// TwinCAT 3 PLC project CollectionTests
// ProgramVersion: 3.1.4026.19
// libraries:
//   AbstractObjectTestLib, * (ekvip automation GmbH)
//   CNM_AbstractObject, * (ekvip automation GmbH)
//   CNM_CollectionInterfaces, * (ekvip automation GmbH)
//   CNM_Collections, * (ekvip automation GmbH)
//   CNM_CollectionTestLib, * (ekvip automation GmbH)
//   CNM_ReturnTypes, * (ekvip automation GmbH)
//   Tc2_Standard, * (Beckhoff Automation GmbH)
//   Tc2_System, * (Beckhoff Automation GmbH)
//   Tc3_Module, * (Beckhoff Automation GmbH)
//   TcUnit, * (www.tcunit.org)
// project tree:
//   / PlcTask.TcTTO
//   POUs/ArrayListSorter/ ContainerBasedArrayListSorterTest.TcPOU, TestArrayList.TcPOU
//   POUs/BBSTrees/ concretBBSTreeTest.TcPOU, TreeTestClass.TcPOU
//   POUs/LinkedList/ LinkedListTest.TcPOU, TestLinkedList.TcPOU
//   POUs/ MAIN.TcPOU
// real-time tasks:
//   TASK PlcTask: cycle T#100us, priority 20, ADS port 350

CONFIGURATION CollectionTests
    RESOURCE PLC ON TwinCAT3
        TASK PlcTask(INTERVAL := T#100us, PRIORITY := 20);
        PROGRAM MAIN WITH PlcTask : MAIN;
    END_RESOURCE
END_CONFIGURATION

// ---- POUs/MAIN.TcPOU
PROGRAM MAIN
VAR
	optionVerbose 						:BOOL := FALSE;
    testCollectionFactory 				:CNM_Collections.CollectionFactory();
	
	
	(*Linked List Tests*)
	linkedList 							:CNM_Collections.LinkedList();
	linkedList2 						:CNM_Collections.LinkedList();
	linkedList3							:CNM_Collections.LinkedList();
	LinkedListTest 						:CNM_CollectionTestLib.ListInterfaceTest(linkedList, linkedList2, testCollectionFactory);
	linkedListDispatcher				:CNM_CollectionTestLib.ListDispatcher(linkedList3);
	linkedListCollectionTest			:CNM_CollectionTestLib.CollectionInterfaceTest(linkedList3, testCollectionFactory, linkedListDispatcher);
	LinkedListObjectTest  				:AbstractObject_Test(linkedList, linkedList2);
	LinkedListTest2						:LinkedListTest(linkedList, linkedList2, testCollectionFactory);
	linkedListForIteratorTest			:CNM_Collections.LinkedList();
	forwardLinkedListIterator			:CNM_Collections.ForwardLinkedListIterator(list:=linkedListForIteratorTest);
	inverseLinkedListIterator			:CNM_Collections.InverseLinkedListIterator(list:=linkedListForIteratorTest);
	linkedListDispatcherIteratorTest	:CNM_CollectionTestLib.ListDispatcher(linkedListForIteratorTest);
	linkedListForwardIteratorTest		:CNM_CollectionTestLib.IteratorInterfaceTest(linkedListForIteratorTest,forwardLinkedListIterator,linkedListDispatcherIteratorTest);
	linkedListInverseIteratorTest		:CNM_CollectionTestLib.IteratorInterfaceTest(linkedListForIteratorTest,inverseLinkedListIterator,linkedListDispatcherIteratorTest);
	
	(*Linkedlistsorter Tests*)
	(*Mergesorter*)
	LinkedListMergeSorter1				:CNM_Collections.LinkedListMergeSorter();
	LinkedListMergeSorter2				:CNM_Collections.LinkedListMergeSorter();
	LinkedListMergeSorterTest			:CNM_CollectionTestLib.ListSorterTest(ListFactory := testCollectionFactory, externListSorter := LinkedListMergeSorter1, verboseLogging := optionVerbose);
	LinkedListMergeSorterObjectTest 	:AbstractObject_Test(LinkedListMergeSorter1, LinkedListMergeSorter2);
	
	(*Array List Tests*)
	arrayList1 							:CNM_Collections.ArrayList();
	arrayList2 							:CNM_Collections.ArrayList();
	arrayList3 							:CNM_Collections.ArrayList();	
	arrayList4							:CNM_Collections.ArrayList();
	ArrayListTest 						:CNM_CollectionTestLib.ListInterfaceTest(arrayList1, arrayList2, testCollectionFactory);
	arrayListDispatcher					:CNM_CollectionTestLib.ListDispatcher(arrayList3);		
	arrayListCollectionTest				:CNM_CollectionTestLib.CollectionInterfaceTest(arrayList3, testCollectionFactory, arrayListDispatcher);
	arrayListIndexableTest 				:CNM_CollectionTestLib.IndexableCollectionTest(arrayList4);
	arrayListObjectTest  				:AbstractObject_Test(arrayList1, arrayList2);
	arrayListForIteratorTest			:CNM_Collections.ArrayList();
	forwardArrayListIterator			:CNM_Collections.ForwardArrayListIterator(arrayList:=arrayListForIteratorTest);
	inverseArrayListIterator			:CNM_Collections.InverseArrayListIterator(arrayList:=arrayListForIteratorTest);
	arrayListDispatcherIteratorTest		:CNM_CollectionTestLib.ListDispatcher(arrayListForIteratorTest);
	arrayListForwardIteratorTest		:CNM_CollectionTestLib.IteratorInterfaceTest(arrayListForIteratorTest,forwardArrayListIterator,arrayListDispatcherIteratorTest);
	arrayListInverseIteratorTest		:CNM_CollectionTestLib.IteratorInterfaceTest(arrayListForIteratorTest,inverseArrayListIterator,arrayListDispatcherIteratorTest);
	
	(*Arraylistsorter Tests*)
	(*Mergesorter*)
	ArrayListMergeSorter1 				:CNM_Collections.ArrayListMergeSorter();
	ArrayListMergeSorter2 				:CNM_Collections.ArrayListMergeSorter();
	ArrayListMergeSorterTest 			:ContainerBasedArrayListSorterTest(ListFactory := testCollectionFactory, externListSorter := ArrayListMergeSorter1, verboseLogging := optionVerbose);
	ArrayListMergeSorterObjectTest 		:AbstractObject_Test(ArrayListMergeSorter1, ArrayListMergeSorter2);
	
	(*Timsorter*)
	ArrayListTwinSorter 				:CNM_Collections.ArrayListTwinSorter();
	ArrayListTwinSorter2 				:CNM_Collections.ArrayListTwinSorter(); 
	ArrayListTwinSorterTest 				:ContainerBasedArrayListSorterTest(ListFactory:=testCollectionFactory,externListSorter := ArrayListTwinSorter, verboseLogging := optionVerbose);
	ArrayListTwinSorterObjectTest 		:AbstractObjectTestLib.AbstractObject_Test(ArrayListTwinSorter, ArrayListTwinSorter2);
	
	(*Shellsorter*)
	ArrayListShellSorter 				:CNM_Collections.ArrayListShellSorter;
	ArrayListShellSorter2 				:CNM_Collections.ArrayListShellSorter;
	ArrayListShellSorterTest 			:ContainerBasedArrayListSorterTest(ListFactory:=testCollectionFactory,externListSorter := ArrayListShellSorter, verboseLogging := optionVerbose);
	ArrayListShellSorterObjectTest 		:AbstractObjectTestLib.AbstractObject_Test(ArrayListShellSorter, ArrayListShellSorter2);

	(*Treetests*)
	TreeFactory							:CNM_Collections.CollectionFactory();
	InterfaceTreeTest					:CNM_CollectionTestLib.BalancedBinaryTreeTest(Treefactory := Treefactory);
	ClassTreeTest						:concretBBSTreeTest(Treefactory := TreeFactory);
	tree1								:CNM_Collections.BalancedBinarySearchTree(0);
	tree2								:CNM_Collections.BalancedBinarySearchTree(0);
	tree3								:CNM_Collections.BalancedBinarySearchTree(0);
	treeDispatcher						:CNM_CollectionTestLib.TreeDispatcher(tree3);
	treeCollectionTest					:CNM_CollectionTestLib.CollectionInterfaceTest(tree3, treeFactory, treeDispatcher);
	objectTreeTest						:AbstractObject_Test(tree1, tree2);
	treeForIteratorTest					:CNM_Collections.BalancedBinarySearchTree(0);
	bfsTreeIterator						:CNM_Collections.BfsBbstIterator(tree:=treeForIteratorTest);
	dfsTreeIterator						:CNM_Collections.DfsBbstIterator(tree:=treeForIteratorTest);
	inorderTreeIterator					:CNM_Collections.InorderBbstIterator(tree:=treeForIteratorTest);
	treeDispatcherIteratorTest			:CNM_CollectionTestLib.TreeDispatcher(treeForIteratorTest);
	treeBFSIteratorTest					:CNM_CollectionTestLib.IteratorInterfaceTest(treeForIteratorTest,bfsTreeIterator,treeDispatcherIteratorTest);
	treeDFSIteratorTest					:CNM_CollectionTestLib.IteratorInterfaceTest(treeForIteratorTest,dfsTreeIterator,treeDispatcherIteratorTest);
	treeInorderIteratorTest				:CNM_CollectionTestLib.IteratorInterfaceTest(treeForIteratorTest,inorderTreeIterator,treeDispatcherIteratorTest);
END_VAR
VAR CONSTANT
	NOT_DEFINED 						:__XWORD := 0;
END_VAR

 TcUnit.RUN_IN_SEQUENCE();

END_PROGRAM

// ---- POUs/LinkedList/LinkedListTest.TcPOU
FUNCTION_BLOCK LinkedListTest EXTENDS CNM_CollectionTestLib.ListInterfaceTest;
VAR_INPUT
END_VAR
VAR_OUTPUT
END_VAR
VAR
END_VAR

THIS^.SortAndCheckPreviousElement('SortAndCheckElementPrevious');

METHOD FB_init : BOOL
VAR_INPUT
    bInitRetains : BOOL; // if TRUE, the retain variables are initialized (warm start / cold start)
    bInCopyCode : BOOL;  // if TRUE, the instance afterwards gets moved into the copy code (online change)
	(*main list to be tested*)
	emptyList1 :CNM_CollectionInterfaces.IList;
	(*secondary list to be tested for appendCollection test*)
	emptyList2 :CNM_CollectionInterfaces.IList;
	(*factory needed for forEach tests, not tested*)
	actionListFactory :CNM_CollectionInterfaces.ICollectionFactory;
END_VAR
THIS^.externalList := emptyList1;
THIS^.externalList2 := emptyList2;
THIS^.listFactory := actionListFactory;
END_METHOD

METHOD SortAndCheckPreviousElement
VAR_INPUT
	testInstanceIdentifier	:STRING(255);
END_VAR
VAR
	testname				:STRING(255);
	dequeuedElement			:CNM_AbstractObject.IObject;
	lastElement				:CNM_CollectionInterfaces.IDoublyLinkedElement;
	lastElementPrevious		:CNM_AbstractObject.IObject;
	foo						:CNM_AbstractObject.IObject;
	comparisonResult		:BOOL;
	index					:INT;
END_VAR
VAR_INST
	newLinkedList			:CNM_CollectionInterfaces.ILinkedList;
	specialList				:TestLinkedList;
	listToSort 				:CNM_CollectionInterfaces.IList;
	sortState				:CNM_ReturnTypes.SingleExecutionState;
	sortReady				:BOOL := FALSE;
	initSuccess				:BOOL := FALSE;
END_VAR
testname := Tc2_Standard.CONCAT('SortAndCheckElementPrevious', testInstanceIdentifier);
IF TcUnit.TEST_ORDERED(testname) THEN
	IF NOT initSuccess THEN
		IF (listFactory.getNewLinkedList(list => newLinkedList) <> CNM_ReturnTypes.SingleExecutionResult.SUCCESS) THEN
			THIS^.AssertTrue(FALSE, 'Creation of linkedList has failed, test has failed');
			TcUnit.TEST_FINISHED();
			RETURN;
		ELSE
			listToSort := newLinkedList;
		END_IF
		FOR index := 0 TO 999 BY 1 DO
			foo := testobjectfactory.getNewTestObject(index);
			listToSort.prepend(foo);
			specialList.prepend(foo);
		END_FOR
		listToSort.sort.ascending(FALSE);
		initSuccess := TRUE;
	END_IF
	IF initSuccess AND_THEN listToSort.sort.ascending(TRUE) = CNM_ReturnTypes.SingleExecutionState.SUCCESS AND sortReady = FALSE THEN
		sortReady := TRUE;
	END_IF
	IF sortReady = TRUE THEN
		dequeuedElement := listToSort.dequeue();
		dequeuedElement.destruct();
		FOR index := 0 TO 998 BY 1 DO
			dequeuedElement := listToSort.dequeue();
			lastElement := specialList.getLastElement;
			lastElementPrevious	:= lastElement.previous.object;
			comparisonResult := lastElementPrevious.isEqual(dequeuedElement);
			IF comparisonResult = FALSE THEN
				AssertFalse(Condition := TRUE, 'the previous element in the list doesn$'t match the element in the special list');
			END_IF
			dequeuedElement.destruct();
			specialList.pop();
		END_FOR
		listToSort.deepDestruct();
		TEST_FINISHED();
	END_IF
END_IF
END_METHOD

END_FUNCTION_BLOCK

// ---- POUs/LinkedList/TestLinkedList.TcPOU
FUNCTION_BLOCK TestLinkedList EXTENDS CNM_Collections.LinkedList
VAR_INPUT
END_VAR
VAR_OUTPUT
END_VAR
VAR
END_VAR

PROPERTY getLastElement : CNM_CollectionInterfaces.IDoublyLinkedElement
GET
getLastElement := THIS^.lastElement;
END_GET
END_PROPERTY

END_FUNCTION_BLOCK

// ---- POUs/ArrayListSorter/ContainerBasedArrayListSorterTest.TcPOU
FUNCTION_BLOCK ContainerBasedArrayListSorterTest EXTENDS CNM_CollectionTestLib.ListSorterTest
VAR_INPUT
END_VAR
VAR_OUTPUT
END_VAR
VAR
	arrayListSorter :CNM_CollectionInterfaces.IArrayListSorter;
END_VAR

SUPER^();
__QUERYINTERFACE(THIS^.Sorter,arrayListSorter);
THIS^.sortAndRescale(
	valuesToSort := RANDOM_1000_INIT,
	sorterToTest := arrayListSorter,
	testInstanceIdentifier:='randomListRescale',
	verboseLogging := THIS^.verboseLogging
);


(*

short summary
=================
Tests that sorting still works correctly, when the container is increased

.. <legal notes>

legal notes
=================
| SPDX-FileCopyrightText: © 2022 ekvip automation GmbH <info@ekvip.de>
| SPDX-License-Identifier: Apache-2.0
| For details check: Apache-2.0_

.. _Apache-2.0: https://www.apache.org/licenses/LICENSE-2.0

.. </legal notes>

parameters
=========================

*)

METHOD sortAndRescale
VAR_INPUT
	(*the Identifier for the test*)
	testInstanceIdentifier	:STRING(255);
	(*The sorter that should be tested*)
	sorterToTest			:CNM_CollectionInterfaces.IArrayListSorter;
	(*Should be true when verbose messages should be printed (for example needed cycles)*)
	verboseLogging			:BOOL;
END_VAR
VAR_IN_OUT
	(*The values that should be sorted*)
	valuesToSort 			:ARRAY[*] OF INT;
END_VAR
VAR_OUTPUT
	(*True when sort is done*)
	finishedSort 			:BOOL;
	(*The amount of cycles used to sort the list*)
	usedCycles 				:INT;
END_VAR
VAR
	testname 				:STRING(255);
	sorterName				:STRING(255);
END_VAR
VAR_INST
	sortableList			:TestArrayList();
	initTest 				:BOOL		:= TRUE; 
	sortDone				:BOOL		:= FALSE;
	cyclesTaken				:INT		:= 0;
	evaluateResults			:BOOL		:= FALSE;
	sortState				:CNM_ReturnTypes.SingleExecutionState;
	listExtended			:BOOL		:= FALSE;
	initialContainerSize	:__XWORD	:= 0;
END_VAR
sorterName := SEL(THIS^.listFactory.isObjectValid(sorter),'internalSorter',Sorter.className);
testname := Tc2_Standard.CONCAT('sortAndRescale.',Tc2_Standard.CONCAT(sorterName, Tc2_Standard.CONCAT('.',testInstanceIdentifier)));
IF TEST_ORDERED(testname) THEN
	IF initTest THEN
		IF THIS^.listFactory.isObjectNull(sorter) THEN
			//test does not work with internal sorter
			TcUnit.TEST_FINISHED();
			RETURN;
		END_IF
		//pretest
		initTest := FALSE;
		listExtended := FALSE;
		cyclesTaken := 0;
		appendArrayToList(listToInit := sortableList,initValues := valuesToSort);
		sortableList.setSorter(sorterToTest);
		sortState := sortableList.sort.ascending(FALSE);
		initialContainerSize := sortableList.currentContainerSize;
		sortDone := FALSE;
		finishedSort := sortDone;
			
	ELSE
		
		//executeTest
		
		sortDone := FALSE;
		finishedSort := sortDone;
		IF NOT ((sortState := sortablelist.sort.ascending(TRUE)) = CNM_ReturnTypes.SingleExecutionState.SUCCESS) THEN 
			cyclesTaken := cyclesTaken + 1;
		END_IF;
		IF sortState = CNM_ReturnTypes.SingleExecutionState.SUCCESS AND NOT listExtended THEN
			WHILE sortableList.currentContainerSize = initialContainerSize DO
				appendArrayToList(listToInit:= sortableList,initValues := valuesToSort);
				sortableList.sort.ascending(FALSE);
			END_WHILE
			listExtended := TRUE;
			sortState := CNM_ReturnTypes.SingleExecutionState.BUSY;
		END_IF
		usedCycles := cyclesTaken;
		finishedSort := sortDone;
		IF sorter.isObjectValid(sortableList) THEN
			IF sortState = CNM_ReturnTypes.SingleExecutionState.SUCCESS THEN 
				//The test is finished within the method "checkIfListSorted".
				checkIfListSorted(initTest := initTest, testname := testname, sortDone := sortDone, cyclesTaken := cyclesTaken, sortableList := sortableList, comparator := 0);
				finishedSort := sortDone;
			ELSIF NOT (sortState = CNM_ReturnTypes.SingleExecutionState.BUSY) THEN
				ASSERTTRUE(FALSE,'sorting ended with unsuspected executionstate'); 
				Test_finished();
				sortableList.deepDestruct();	
				initTest := TRUE;
				RETURN;
			END_IF
		ELSE
			Test_finished();
			sortableList.deepDestruct();	
			initTest := TRUE;
			RETURN;
		END_IF
	END_IF
END_IF
END_METHOD

END_FUNCTION_BLOCK

// ---- POUs/ArrayListSorter/TestArrayList.TcPOU
FUNCTION_BLOCK TestArrayList EXTENDS CNM_Collections.ArrayList
VAR_INPUT
END_VAR
VAR_OUTPUT
END_VAR
VAR
END_VAR

PROPERTY currentContainerSize : __XWORD
GET
currentContainerSize := THIS^.currentContainerCapacity;
END_GET
END_PROPERTY

END_FUNCTION_BLOCK

// ---- POUs/BBSTrees/concretBBSTreeTest.TcPOU
(*

short summary
=================
A functionblock to test the concrete Treeimplementation from the CNM_Collections Library. 
These tests are dependend on the implementations, since they check the rotations that are performed during insert and remove.
Other implementation independed tests can be found in the CNM_Collection_TestLib

.. <legal notes>

legal notes
=================
| SPDX-FileCopyrightText: © 2023 ekvip automation GmbH <info@ekvip.de>
| SPDX-License-Identifier: Apache-2.0
| For details check: Apache-2.0_

.. _Apache-2.0: https://www.apache.org/licenses/LICENSE-2.0

.. </legal notes>

parameters
=========================

*)
FUNCTION_BLOCK concretBBSTreeTest EXTENDS TcUnit.FB_TestSuite
VAR_INPUT
END_VAR
VAR_OUTPUT
END_VAR
VAR
	treeFactory 		:CNM_CollectionInterfaces.ICollectionFactory;
	testObjectFactory	:CNM_CollectionTestLib.testObjectFactory;
END_VAR

THIS^.insertElementInEmptyTree('');
THIS^.removeElements('');
THIS^.insertElementsToCheckRotation('');
THIS^.nodesAreInCorrectOrderWithReverseOrderComparator('');

METHOD checkNodeReverseOrder : BOOL
VAR_INPUT
	currentNode						:CNM_CollectionInterfaces.IBinaryTreeNode;
END_VAR
VAR
	comparator						:CNM_CollectionTestLib.ReverseOrderComparator;
    leftGreater 					:BOOL;
    rightGreater					:BOOL;
END_VAR
VAR_IN_OUT
	leftChildsCurrentNode			:CNM_CollectionInterfaces.IBinaryTreeNode;
	rightChildsCurrentNode			:CNM_CollectionInterfaces.IBinaryTreeNode;
END_VAR
IF currentNode = 0 THEN
	// An empty node is considered valid
	checkNodeReverseOrder := TRUE;
	RETURN;
END_IF
    
// Initialize children validity
leftGreater := TRUE;
rightGreater := TRUE;

// Check the left child
IF currentNode.leftChild <> 0 THEN
	IF comparator.compare(currentNode.leftChild, currentNode) = CNM_ReturnTypes.ComparationResult.GREATER THEN
		leftGreater := FALSE;
		leftChildsCurrentNode := currentNode;
	ELSE
		leftGreater := THIS^.checkNodeReverseOrder(currentNode.leftChild, leftChildsCurrentNode, rightChildsCurrentNode);
	END_IF
END_IF

// Check the right child
IF currentNode.rightChild <> 0 THEN
	IF comparator.compare(currentNode.rightChild, currentNode) = CNM_ReturnTypes.ComparationResult.SMALLER THEN
		rightGreater := FALSE;
		rightChildsCurrentNode := currentNode;
	ELSE
		rightGreater := THIS^.checkNodeReverseOrder(currentNode.rightChild, leftChildsCurrentNode, rightChildsCurrentNode);
	END_IF
END_IF

checkNodeReverseOrder := leftGreater AND rightGreater;
END_METHOD

(*

short summary
=================
function to create a new balanced binary searchtree node

.. <legal notes>

legal notes
=================
| SPDX-FileCopyrightText: © 2023 ekvip automation GmbH <info@ekvip.de>
| SPDX-License-Identifier: Apache-2.0
| For details check: Apache-2.0_

.. _Apache-2.0: https://www.apache.org/licenses/LICENSE-2.0

.. </legal notes>

parameters
=========================

*)
METHOD FB_init :BOOL
VAR_INPUT
    bInitRetains 	:BOOL; // if TRUE, the retain variables are initialized (warm start / cold start)
    bInCopyCode		:BOOL;  // if TRUE, the instance afterwards gets moved into the copy code (online change)
	(*The factory that is used to instantiate new trees*)
	Treefactory 	:CNM_CollectionInterfaces.ICollectionFactory;
END_VAR
THIS^.treefactory := Treefactory;
END_METHOD

(*

short summary
=================
helperfunction that creates the full testmessage

.. <legal notes>

legal notes
=================
| SPDX-FileCopyrightText: © 2023 ekvip automation GmbH <info@ekvip.de>
| SPDX-License-Identifier: Apache-2.0
| For details check: Apache-2.0_

.. _Apache-2.0: https://www.apache.org/licenses/LICENSE-2.0

.. </legal notes>

parameters
=========================
:return: the complete Testmessage
*)
METHOD generateTestmessage :STRING
VAR_INPUT
	(*The name of the test*)
	name :STRING(255);
	(*The message that should be printed*)
	msg :STRING; 
END_VAR
generateTestmessage := CONCAT((CONCAT('For Test: ',name)),msg);
END_METHOD

(*

short summary
=================
Test that 
- tries to insert a null object and assumes that it fails (no null objects are allowed in collections)
- checks that the root of an empty tree is null 
- and that the insert of a single insert is a success and the root now contains this element

.. <legal notes>

legal notes
=================
| SPDX-FileCopyrightText: © 2023 ekvip automation GmbH <info@ekvip.de>
| SPDX-License-Identifier: Apache-2.0
| For details check: Apache-2.0_

.. _Apache-2.0: https://www.apache.org/licenses/LICENSE-2.0

.. </legal notes>

parameters
=========================

*)

METHOD insertElementInEmptyTree
VAR_INPUT
	(*unique Identifier for each instance to differentiate between multiple instances*)
	testInstanceIdentifier 	:STRING(255);
END_VAR
VAR
	tree 					:TreeTestClass(OBJECT_NOT_REFERENCED);
	treePointer 			:POINTER TO CNM_Collections.BalancedBinarySearchTree;
	testname				:STRING(255);
	newnode 				:CNM_AbstractObject.IObject;
END_VAR
VAR CONSTANT
	{attribute 'suppress_warning_0' := 'C0228'}
	OBJECT_NOT_REFERENCED 	:__XWORD	:= 0;
	{attribute 'restore_warning_0' := 'C0228'}
END_VAR
testname := CONCAT('insertInEmptyTree',testInstanceIdentifier);
IF TEST_ORDERED(testname) THEN 
	AssertTrue(tree.tree.insert(newnode) = CNM_ReturnTypes.SingleExecutionResult.ABORTED,generateTestmessage(testInstanceIdentifier,'insert of an null object didnt return ABORTED as expected'));
	newnode := THIS^.testobjectfactory.getNewTestObject(value:=2);
	
	//Asserts
	AssertTrue(Condition := newnode.isObjectNull(tree.testRootNode) , generateTestmessage(name:=testInstanceIdentifier,msg:='the testRootNode of the empty tree where not null'));
	ASSERTTRUE(tree.tree.insert(object:=newnode)=CNM_ReturnTypes.SingleExecutionResult.SUCCESS, generateTestmessage(name := testInstanceIdentifier, msg := 'inserting of Node Fooobject(2) failed'));
	IF  newnode.isObjectNull(tree.testRootNode) THEN
		AssertFalse(Condition :=TRUE, generateTestmessage(name := testInstanceIdentifier, msg :='after insert an object, the testRootNode was still null'));
		TEST_FINISHED();
		RETURN;
	END_IF;
	AssertTrue(Condition := tree.testRootNode.object.isEqual(newNode), generateTestmessage(name := testInstanceIdentifier, 'after inserting root wasn$'t the object that was inserted'));
	TEST_FINISHED();
	IF tree.isObjectValid(newNode) THEN
		newNode.deepDestruct();
	END_IF
END_IF
END_METHOD

(*

short summary
=================
Test that checks if the rotations used for balancing are performed correct during insert of elements.

.. <legal notes>

legal notes
=================
| SPDX-FileCopyrightText: © 2023 ekvip automation GmbH <info@ekvip.de>
| SPDX-License-Identifier: Apache-2.0
| For details check: Apache-2.0_

.. _Apache-2.0: https://www.apache.org/licenses/LICENSE-2.0

.. </legal notes>

parameters
=========================

*)

METHOD insertElementsToCheckRotation
VAR_INPUT
	(*The identifier used to differentiate between mutliple instances of this test*)
	testInstanceIdentifier 	:STRING(255);
END_VAR
VAR
	tree 					:TreeTestClass(OBJECT_NOT_REFERENCED);
	testname				:STRING(255);
	node10 					:CNM_AbstractObject.IObject;
	node20 					:CNM_AbstractObject.IObject;
	node4 					:CNM_AbstractObject.IObject;
	node15 					:CNM_AbstractObject.IObject;
	node17 					:CNM_AbstractObject.IObject;
	node3 					:CNM_AbstractObject.IObject;
	node2 					:CNM_AbstractObject.IObject;
	node1 					:CNM_AbstractObject.IObject;
	iterateObject 			:CNM_AbstractObject.IObject;
	rootNode 				:POINTER TO CNM_CollectionTestLib.testObject;
	binaryRoot 				:CNM_CollectionInterfaces.IBinaryTreeNode;
	rootNodeOrderValue 		:INT;
	iterator				:CNM_CollectionInterfaces.IIterator;
END_VAR
VAR CONSTANT
	{attribute 'suppress_warning_0' := 'C0228'}
	OBJECT_NOT_REFERENCED 	:__XWORD 	:= 0;
	{attribute 'restore_warning_0' := 'C0228'}
END_VAR
testname := CONCAT('TreeCheckRotation',testInstanceIdentifier);
IF TEST_ORDERED(testname)  THEN 
	//pre test
	node10 := THIS^.testobjectfactory.getNewTestObject(value:=10);
	node20 := THIS^.testobjectfactory.getNewTestObject(value:=20);
	node4 := THIS^.testobjectfactory.getNewTestObject(value:=4);
	node15 := THIS^.testobjectfactory.getNewTestObject(value:=15);
	node17 := THIS^.testobjectfactory.getNewTestObject(value:=17);
	node3 := THIS^.testobjectfactory.getNewTestObject(3);
	node2 := THIS^.testobjectfactory.getNewTestObject(2);
	node1 := THIS^.testobjectfactory.getNewTestObject(1);
	AssertTrue(tree.tree.insert(node2)=CNM_ReturnTypes.SingleExecutionResult.SUCCESS, generateTestmessage(name := testname, msg := 'inserting of not existing Node Fooobject(2) failed'));
	AssertTrue(tree.tree.insert(node1)=CNM_ReturnTypes.SingleExecutionResult.SUCCESS, generateTestmessage(name := testname, msg := 'inserting of not existing Node Fooobject(1) failed'));
	AssertTrue(tree.tree.insert(node3)=CNM_ReturnTypes.SingleExecutionResult.SUCCESS, generateTestmessage(name := testname, msg := 'inserting of not existing Node Fooobject(3) failed'));
	AssertTrue(tree.tree.insert(node10)=CNM_ReturnTypes.SingleExecutionResult.SUCCESS, generateTestmessage(name := testname, msg := 'inserting of not existing Node Fooobject(10) failed'));
	AssertTrue(tree.tree.insert(node20)=CNM_ReturnTypes.SingleExecutionResult.SUCCESS, generateTestmessage(name := testname, msg := 'inserting of not existing Node Fooobject(20) failed'));
	__QUERYINTERFACE(tree.testRootNode,binaryroot);
	//LeftRotation Expected
		IF tree.isObjectNull(binaryroot.rightChild) THEN 
			AssertFalse(Condition := TRUE, generateTestmessage(name := testname, msg :='after insert an object greater than root, root.rightChild was still null'));
			TEST_FINISHED();
			RETURN;	
		END_IF
		AssertTrue(Condition := binaryRoot.rightChild.object = node10, Message:='after LRotation the rotroot wasnt what was exp(10)');
		AssertTrue(Condition := binaryRoot.rightChild.leftChild.object = node3, Message:='after LRotation the rotroot.lchild wasnt what was exp(3)');
		AssertTrue(Condition := binaryRoot.rightChild.rightChild.object = node20, Message:='after LRotation the rotroot.rchild wasnt what was exp(20)');
	AssertTrue(tree.tree.insert(node4)=CNM_ReturnTypes.SingleExecutionResult.SUCCESS, generateTestmessage(name := testname, msg := 'inserting of not existing Node Fooobject(4) failed'));
	AssertTrue(tree.tree.insert(node17)=CNM_ReturnTypes.SingleExecutionResult.SUCCESS, generateTestmessage(name := testname, msg := 'inserting of not existing Node Fooobject(17) failed'));
	AssertTrue(tree.tree.insert(node15)=CNM_ReturnTypes.SingleExecutionResult.SUCCESS, generateTestmessage(name := testname, msg := 'inserting of not existing Node Fooobject(15) failed'));
	
	//requery treenode because it should have changed due to rotation
	__QUERYINTERFACE(tree.testRootNode,binaryRoot);
	
	IF node10.isObjectNull(binaryroot) THEN 
			AssertFalse(Condition := TRUE, generateTestmessage(name := testname, msg :='root was unexpected null'));
			TEST_FINISHED();
			RETURN;	
	END_IF
		AssertTrue(Condition := binaryRoot.object = node3, Message:='after DRotation the root wasnt what was exp(3)');
	//at this point it is sure that binaryroot is unequal zero

	IF binaryRoot.isObjectNull(binaryroot.leftChild) THEN
			AssertFalse(Condition := TRUE, generateTestmessage(name := testname, msg :='root.left was unexpected null'));
			TEST_FINISHED();
			RETURN;	
	END_IF
	AssertTrue(Condition := binaryRoot.leftChild.object = node2, generateTestmessage(name := testname, msg := 'after DRotation, root.left wasnt exp(2)'));
	
	IF binaryRoot.isObjectNull(binaryroot.leftChild.leftChild) THEN
			AssertFalse(Condition := TRUE, generateTestmessage(name := testname, msg :='root.left.left was unexpected null'));
			TEST_FINISHED();
			RETURN;	
	END_IF
	AssertTrue(Condition := binaryRoot.leftChild.leftChild.object = node1, generateTestmessage(name := testname, msg := 'after DRotation, root.left.left wasnt exp(1)'));
	
	IF binaryRoot.isObjectNull(binaryroot.rightChild) THEN
			AssertFalse(Condition := TRUE, generateTestmessage(name := testname, msg :='root.right was unexpected null'));
			TEST_FINISHED();
			RETURN;	
	END_IF
	AssertTrue(Condition := binaryRoot.rightChild.object = node10, generateTestmessage(name := testname, msg := 'after DRotation, root.right wasnt exp(10)'));
	
	IF binaryRoot.isObjectNull(binaryroot.rightChild.leftChild) THEN
			AssertFalse(Condition := TRUE, generateTestmessage(name := testname, msg :='root.right.left was unexpected null'));
			TEST_FINISHED();
			RETURN;	
	END_IF
	AssertTrue(Condition := binaryRoot.rightChild.leftChild.object = node4, generateTestmessage(name := testname, msg := 'after DRotation, root.right.left wasnt exp(4)'));
		
	IF binaryRoot.isObjectNull(binaryroot.rightChild.rightChild) THEN
			AssertFalse(Condition := TRUE, generateTestmessage(name := testname, msg :='root.right.right was unexpected null'));
			TEST_FINISHED();
			RETURN;	
	END_IF
	AssertTrue(Condition := binaryRoot.rightChild.rightChild.object = node17, generateTestmessage(name := testname, msg := 'after RRotation, root.right.right wasnt exp(17)'));
	
	IF binaryRoot.isObjectNull(binaryroot.rightChild.rightChild.leftChild) THEN
			AssertFalse(Condition := TRUE, generateTestmessage(name := testname, msg :='root.right.right.left was unexpected null'));
			TEST_FINISHED();
			RETURN;	
	END_IF
	AssertTrue(Condition := binaryRoot.rightChild.rightChild.leftChild.object = node15, generateTestmessage(name := testname, msg := 'after RRotation, root.right.right.left wasnt exp(15)'));
	
	IF binaryRoot.isObjectNull(binaryroot.rightChild.rightChild.rightChild) THEN
			AssertFalse(Condition := TRUE, generateTestmessage(name := testname, msg :='root.right.right.right was unexpected null'));
			TEST_FINISHED();
			RETURN;	
	END_IF
	AssertTrue(Condition := binaryRoot.rightChild.rightChild.rightChild.object = node20, generateTestmessage(name := testname, msg := 'after RRotation, root.right.right.right wasnt exp(20)'));
	//Test that leafs are true leafs and have no childs
	ASSERTTRUE(Condition := binaryroot.isObjectNull(binaryroot.leftChild.leftChild.leftChild), Message:=generateTestmessage(name:=testname, msg := 'leaf(1) leftchild was not null'));
	ASSERTTRUE(Condition := binaryroot.isObjectNull(binaryroot.leftChild.leftChild.rightChild), Message:=generateTestmessage(name:=testname, msg := 'leaf(1) rightchild was not null'));	
	ASSERTTRUE(Condition := binaryroot.isObjectNull(binaryroot.leftChild.rightChild), Message:=generateTestmessage(name:=testname, msg := 'leaf(2) rightchild was not null'));
	ASSERTTRUE(Condition := binaryroot.isObjectNull(binaryroot.rightChild.rightChild.leftChild.leftChild), Message:=generateTestmessage(name:=testname, msg := 'leaf(15) leftchild was not null'));
	ASSERTTRUE(Condition := binaryroot.isObjectNull(binaryroot.rightChild.rightChild.leftChild.rightChild), Message:=generateTestmessage(name:=testname, msg := 'leaf(15) rightchild was not null'));
	ASSERTTRUE(Condition := binaryroot.isObjectNull(binaryroot.rightChild.leftChild.leftChild), Message:=generateTestmessage(name:=testname, msg := 'leaf(4) leftchild was not null'));
	ASSERTTRUE(Condition := binaryroot.isObjectNull(binaryroot.rightChild.leftChild.rightChild), Message:=generateTestmessage(name:=testname, msg := 'leaf(4) rightchild was not null'));
	ASSERTTRUE(Condition := binaryroot.isObjectNull(binaryroot.rightChild.rightChild.rightChild.leftChild), Message:=generateTestmessage(name:=testname, msg := 'leaf(20) leftchild was not null'));
	ASSERTTRUE(Condition := binaryroot.isObjectNull(binaryroot.rightChild.rightChild.rightChild.rightChild), Message:=generateTestmessage(name:=testname, msg := 'leaf(20) rightChild was not null'));
	//Test Treesize
	AssertEquals_LWORD(Expected := 8,Actual := tree.size,Message := generateTestmessage(name := testname, msg := 'treesize wasnt correct after insert'));
	//Test the containsObject 
	ASSERTTRUE(Condition := tree.containsObject(object := node10), Message := generateTestmessage(name := testname, msg := 'containsObject(10) failed for existing node'));
	ASSERTTRUE(Condition := tree.containsObject(object := node20), Message := generateTestmessage(name := testname, msg := 'containsObject(20) failed for existing node'));
	ASSERTTRUE(Condition := tree.containsObject(object := node4), Message := generateTestmessage(name := testname, msg := 'containsObject(4) failed for existing node'));
	ASSERTTRUE(Condition := tree.containsObject(object := node15), Message := generateTestmessage(name := testname, msg := 'containsObject(15) failed for existing node'));
	ASSERTTRUE(Condition := tree.containsObject(object := node17), Message := generateTestmessage(name := testname, msg := 'containsObject(17) failed for existing node'));
	ASSERTTRUE(Condition := tree.containsObject(object := node3), Message := generateTestmessage(name := testname, msg := 'containsObject(3) failed for existing node'));
	ASSERTTRUE(Condition := tree.containsObject(object := node2), Message := generateTestmessage(name := testname, msg := 'containsObject(2) failed for existing node'));
	ASSERTTRUE(Condition := tree.containsObject(object := node1), Message := generateTestmessage(name := testname, msg := 'containsObject(1) failed for existing node'));
	//Iterate
	tree.createNewIterator(iterator => iterator);
	iterator.iterate(execute := FALSE);
	iterator.iterate(execute:=TRUE,object => iterateObject);
	ASSERTTRUE(Condition := iterateObject=node1, Message := generateTestmessage(name := testname, msg := 'iterate failed at 1 object'));
	iterator.iterate(execute:=TRUE,object => iterateObject);
	ASSERTTRUE(Condition := iterateObject = node2, Message := generateTestmessage(name := testname, msg := 'iterate failed at 2 object'));
	iterator.iterate(execute:=TRUE,object => iterateObject);
	ASSERTTRUE(Condition := iterateObject = node3, Message := generateTestmessage(name := testname, msg := 'iterate failed at 3 object'));
	iterator.iterate(execute:=TRUE,object => iterateObject);
	ASSERTTRUE(Condition := iterateObject = node4, Message := generateTestmessage(name := testname, msg := 'iterate failed at 4 object'));
	iterator.iterate(execute:=TRUE,object => iterateObject);
	ASSERTTRUE(Condition := iterateObject = node10, Message := generateTestmessage(name := testname, msg := 'iterate failed at 5 object'));
	iterator.iterate(execute:=TRUE,object => iterateObject);
	ASSERTTRUE(Condition := iterateObject = node15, Message := generateTestmessage(name := testname, msg := 'iterate failed at 6 object'));
	iterator.iterate(execute:=TRUE,object => iterateObject);
	ASSERTTRUE(Condition := iterateObject = node17, Message := generateTestmessage(name := testname, msg := 'iterate failed at 7 object'));
	iterator.iterate(execute:=TRUE,object => iterateObject);
	ASSERTTRUE(Condition := iterateObject = node20, Message := generateTestmessage(name := testname, msg := 'iterate failed at 8 object'));      
	iterator.iterate(execute := FALSE); 
	Test_FINISHED();
	//clear tree to free memory captured from nodecontainers
	tree.clear();
	//clear nodecontent
	iterator.destruct();
	node10.destruct();
	node20.destruct();
	node4.destruct();
	node15.destruct();
	node17.destruct();
	node3.destruct();
	node2.destruct();
	node1.destruct();
END_IF
END_METHOD

METHOD nodesAreInCorrectOrderWithReverseOrderComparator
VAR_INPUT
	(*unique Identifier for each instance to differentiate between multiple instances*)
	testInstanceIdentifier 	:Tc2_System.T_MaxString;
	(*The comparator that should be used for the test*)
END_VAR
VAR
	comparator						:CNM_CollectionTestLib.ReverseOrderComparator;
	tree 							:TreeTestClass(comparator);
	testname 						:Tc2_System.T_MaxString;
	nodes 							:ARRAY[0..99] OF CNM_AbstractObject.IObject;
	index 							:INT;
	successfulPass					:BOOL	:= TRUE;
	validityCheckObject				:CNM_AbstractObject.IObject;
	isCorrectlyOrdered				:BOOL	:= FALSE;
	leftChildsCurrentNode			:CNM_CollectionInterfaces.IBinaryTreeNode;
	rightChildsCurrentNode			:CNM_CollectionInterfaces.IBinaryTreeNode;
	leftChildsCurrentNodeObject		:POINTER TO CNM_CollectionTestLib.TestObject;
	leftChildNodeObject				:POINTER TO CNM_CollectionTestLib.TestObject;
	rightChildsCurrentNodeObject	:POINTER TO CNM_CollectionTestLib.TestObject;
	rightChildNodeObject			:POINTER TO CNM_CollectionTestLib.TestObject;
END_VAR
testname := CONCAT('nodesAreInCorrectOrderWithReverseOrderComparator', testInstanceIdentifier);
IF TEST_ORDERED(testname) THEN 
	validityCheckObject := testobjectfactory.getNewTestObject(1);
	successfulPass := TRUE;
	
	FOR index := 0 TO 99 BY 1 DO
		nodes[index] := THIS^.testobjectfactory.getNewTestObject(index);
		successfulPass := (
			successfulPass
			AND (tree.tree.insert(nodes[index]) = CNM_ReturnTypes.SingleExecutionResult.SUCCESS)
		);
		
	END_FOR
	
	IF NOT successfulPass THEN
		AssertTrue(FALSE, 'Inserting nodes to tree has failed, test couldn$'t run');
		JMP testFinished;
	END_IF
	
	isCorrectlyOrdered := checkNodeReverseOrder(tree.testRootNode, leftChildsCurrentNode, rightChildsCurrentNode);
	
	THIS^.AssertTrue(isCorrectlyOrdered, 'Nodes in the tree weren$'t correctly ordered');
	
	IF validityCheckObject.isObjectValid(leftChildsCurrentNode) THEN
		__QUERYPOINTER(leftChildsCurrentNode.object, leftChildsCurrentNodeObject);
		__QUERYPOINTER(leftChildsCurrentNode.leftChild.object, leftChildNodeObject);
		THIS^.AssertTrue(
			FALSE, 
			Tc2_Standard.CONCAT('Left child was smaller at node ', TO_STRING(leftChildsCurrentNodeObject^.orderValue))
		);
		
		THIS^.AssertTrue(
			FALSE, 
			Tc2_Standard.CONCAT('Left child had value ', TO_STRING(leftChildNodeObject^.orderValue))
		);
		
	END_IF
	
	IF validityCheckObject.isObjectValid(rightChildsCurrentNode) THEN
		__QUERYPOINTER(rightChildsCurrentNode.object, rightChildsCurrentNodeObject);
		__QUERYPOINTER(rightChildsCurrentNode.rightChild.object, rightChildNodeObject);
		THIS^.AssertTrue(
			FALSE,
			Tc2_Standard.CONCAT('Right child was greater at node ', TO_STRING(rightChildsCurrentNodeObject^.orderValue))
		);
		
		THIS^.AssertTrue(
			FALSE,
			Tc2_Standard.CONCAT('Right child had value ', TO_STRING(rightChildNodeObject^.orderValue))
		);
		
	END_IF
	
	testFinished:
	tree.deepDestruct();
	validityCheckObject.destruct();
	TEST_FINISHED();
END_IF
END_METHOD

(*

short summary
=================
function to create a new balanced binary searchtree node

.. <legal notes>

legal notes
=================
| SPDX-FileCopyrightText: © 2023 ekvip automation GmbH <info@ekvip.de>
| SPDX-License-Identifier: Apache-2.0
| For details check: Apache-2.0_

.. _Apache-2.0: https://www.apache.org/licenses/LICENSE-2.0

.. </legal notes>

parameters
=========================

*)

METHOD removeElements
VAR_INPUT
(*The identifier used to differentiate between mutliple instances of this test*)	
	testInstanceIdentifier 	:STRING(255);
END_VAR
VAR
	tree 					:TreeTestClass(OBJECT_NOT_REFERENCED);
	testname				:STRING(255);
	nodes 					:ARRAY[0..7] OF CNM_AbstractObject.IObject;
	node17 					:CNM_AbstractObject.IObject;
	node20 					:CNM_AbstractObject.IObject;
	node3 					:CNM_AbstractObject.IObject;
	node10 					:CNM_AbstractObject.IObject;
	node15 					:CNM_AbstractObject.IObject;
	node4 					:CNM_AbstractObject.IObject;
	node2 					:CNM_AbstractObject.IObject;
	node1 					:CNM_AbstractObject.IObject;
	binaryRoot 				:CNM_CollectionInterfaces.IBalancedBinarySearchTreeNode;
	index					:INT := 0;
END_VAR
VAR CONSTANT
	NodeValues 				:ARRAY[0..7] OF INT		:= [2,1,3,10,20,4,17,15];
	{attribute 'suppress_warning_0' := 'C0228'}
	OBJECT_NOT_REFERENCED 	:__XWORD	:= 0;
	{attribute 'restore_warning_0' := 'C0228'}
END_VAR
testname := CONCAT('removeElements',testInstanceIdentifier);
IF TEST_ORDERED(testname) THEN 
	//pre test
	IF __QUERYINTERFACE(tree.testRootNode,binaryRoot) THEN
		FOR index := 0 TO 7 BY 1 DO
			nodes[index] := THIS^.testobjectfactory.getNewTestObject(NodeValues[index]);
			tree.tree.insert(nodes[Index]);
		END_FOR
		node17 := nodes[0];
		node20 := nodes[1];
		node3 := nodes[2];
		node10:= nodes[3];
		node15 := nodes[4];
		node4 := nodes[5];
		node2 := nodes[6];
		node1 := nodes[7];

		//test remove nodes and check after removing them that tree is correct (element is missing / rotation etc was correct 
		ASSERTTRUE(Condition := tree.tree.remove(node20)=CNM_ReturnTypes.SingleExecutionResult.SUCCESS, Message := generateTestmessage(name := testname,msg:='remove of node 20 failed'));
		ASSERTTRUE(Condition := binaryroot.isObjectNull(binaryroot.rightChild.rightChild.rightChild), Message := generateTestmessage(name := testname, msg := 'removed leaf wasnt replaceed with null'));
		ASSERTTRUE(Condition:= tree.tree.remove(node17)=CNM_ReturnTypes.SingleExecutionResult.SUCCESS, Message := generateTestmessage(name:=testname,msg:='remove of node(17) failed'));
 		ASSERTTRUE(Condition := binaryroot.rightChild.rightChild.object = node15, Message := generateTestmessage(name := testname,msg:='removed node(17) wasnt replaced by leftChild'));
		ASSERTTRUE(Condition := tree.tree.remove(node3)=CNM_ReturnTypes.SingleExecutionResult.SUCCESS, Message := generateTestmessage(name:=testname, msg:='remove of rootnode failed'));
		//Tree was rotatet, so get new root
		__QUERYINTERFACE(tree.testRootNode,binaryroot);
		ASSERTTRUE(Condition := binaryroot.object = node4, Message := generateTestmessage(name:=testname, msg:='renoved root wasnt replaced by inorder successor'));
		ASSERTTRUE(Condition := tree.tree.remove(node10)=CNM_ReturnTypes.SingleExecutionResult.SUCCESS, Message := generateTestmessage(name:=testname,msg:='remove of rootnode.right(10) failed'));
		ASSERTTRUE(Condition := binaryRoot.rightChild.object = node15, Message := generateTestmessage(name:=Testname,msg:='removed root.right(10) wasnt replaced with only child(15)'));
		ASSERTTRUE(Condition := tree.tree.remove(node15)=CNM_ReturnTypes.SingleExecutionResult.SUCCESS, Message := generateTestmessage(name := testname, msg := 'remove of root.rightChild failed'));
		//Tree was rotatet so get new root
		__QUERYINTERFACE(tree.testRootNode,binaryroot);
		ASSERTTRUE(Condition := binaryroot.object =  node2, Message := generateTestmessage(name := testname, msg := 'after rotation root wasnt what was expected'));
		ASSERTTRUE(Condition := binaryroot.leftChild.object = node1, Message := generateTestmessage(name := testname, msg := 'after rotation root.left wasnt what was expected'));
		ASSERTTRUE(Condition := binaryroot.rightChild.object = node4, Message := generateTestmessage(name := testname, msg := 'after rotation root.right wasnt what was expected'));
		//Test Treesize
		AssertEquals_LWORD(Expected := 3,Actual := tree.size,Message := generateTestmessage(name := testname, msg := 'treesize wasnt correct after delete'));
		//Test contains element
		ASSERTFALSE(Condition := tree.containsObject(node17),Message := generateTestmessage(name := testname, msg := 'containsObject(17) was true but tree hasnt 17 anymore'));
		ASSERTFALSE(Condition := tree.containsObject(node20),Message := generateTestmessage(name := testname, msg := 'containsObject(20) was true but tree hasnt 20 anymore'));
		ASSERTFALSE(Condition := tree.containsObject(node3),Message := generateTestmessage(name := testname, msg := 'containsObject(3) was true but tree hasnt 3 anymore'));
		ASSERTFALSE(Condition := tree.containsObject(node10),Message := generateTestmessage(name := testname, msg := 'containsObject(10) was true but tree hasnt 10 anymore'));
		ASSERTFALSE(Condition := tree.containsObject(node15),Message := generateTestmessage(name := testname, msg := 'containsObject(15) was true but tree hasnt 15 anymore'));
		ASSERTTRUE(Condition := tree.containsObject(node4),Message := generateTestmessage(name := testname, msg := 'containsObject(4) was flase but tree still has it'));
		ASSERTTRUE(Condition := tree.containsObject(node2),Message := generateTestmessage(name := testname, msg := 'containsObject(2) was flase but tree still has it'));
		ASSERTTRUE(Condition := tree.containsObject(node1),Message := generateTestmessage(name := testname, msg := 'containsObject(1) was flase but tree still has it'));
	
		//clean up the objects that I removed 
		IF tree.isObjectValid(node17) THEN
			node17.destruct();	
		END_IF
		IF tree.isObjectValid(node20) THEN
			node20.destruct();	
		END_IF
		IF tree.isObjectValid(node3) THEN
			node3.destruct();	
		END_IF
		IF tree.isObjectValid(node10) THEN
			node10.destruct();	
		END_IF
		IF tree.isObjectValid(node15) THEN
			node15.destruct();	
		END_IF
		
	END_IF
	
	TEST_FINISHED();
	
	tree.clear();
	FOR index := 0 TO 7 BY 1 DO
		IF tree.isObjectValid(nodes[index]) THEN
			nodes[index].destruct();
		END_IF
	END_FOR
END_IF
END_METHOD

END_FUNCTION_BLOCK

// ---- POUs/BBSTrees/TreeTestClass.TcPOU
FUNCTION_BLOCK TreeTestClass EXTENDS CNM_Collections.BalancedBinarySearchTree
VAR_INPUT
END_VAR
VAR_OUTPUT
END_VAR
VAR
END_VAR

(*

short summary
=================
The constructor ``FB_init`` is needed to create an unique hash code.
The hash code is a pseudo random number create with a xorshift_ algorithm.
It can be overwritten on derivations, because it will be called implicit, ``SUPER^.FB_init()`` is not required.
For more information check: `Behavoir with derived function blocks`_

.. _Behavoir with derived function blocks: https://infosys.beckhoff.com/content/1033/tc3_plc_intro/5482088715.html?id=6983869892358031022

.. _xorshift: https://en.wikipedia.org/wiki/Xorshift

.. <legal notes>

legal notes
=================
| SPDX-FileCopyrightText: © 2022 ekvip automation GmbH <info@ekvip.de>
| SPDX-License-Identifier: Apache-2.0
| For details check: Apache-2.0_

.. _Apache-2.0: https://www.apache.org/licenses/LICENSE-2.0

.. </legal notes>

parameters
=================

*)

METHOD FB_init : BOOL
VAR_INPUT
	(* if TRUE, the retain variables are initialized (warm start / cold start)*)
	bInitRetains	:BOOL;
	(* if TRUE, the instance afterwards gets moved into the copy code (online change) *)
	bInCopyCode		:BOOL;  
	(*Optional comparator*)
	nodeComparator 	:CNM_AbstractObject.IComparator	:= OBJECT_NOT_REFERENCED;
END_VAR
VAR
	{attribute 'hide'}
	newHashstate3		:CNM_AbstractObject.Hashcode;
END_VAR
VAR CONSTANT
	{attribute 'hide'}
	NUMBER_OF_LEFT_SHIFTS		:UINT	:= 17;
	{attribute 'hide'}
	NUMBER_OF_LEFT_ROTATIONS	:UINT   := 45;
	OBJECT_NOT_REFERENCED 		:__XWORD := 0;
END_VAR
THIS^.collectionSize := 0;
THIS^.nodeComparator := nodeComparator;
END_METHOD

PROPERTY PUBLIC testRootNode : CNM_CollectionInterfaces.IBalancedBinarySearchTreeNode
GET
testRootNode := THIS^.rootNode;
END_GET
END_PROPERTY

END_FUNCTION_BLOCK
